(* IEC 61131-3 sources: Industry-PLC-LLM/data/PLCBEAD_repo/PLCBEAD_PLCEmbed-main/PLC-BEAD/Source/GEB/DWORD_OF_BYTE, 1 file *)

(* ---- DWORD_OF_BYTE.ST ---- *)
FUNCTION DWORD_OF_BYTE:DWORD
	VAR_INPUT
		B3 :	BYTE;
		B2 :	BYTE;
		B1 :	BYTE;
		B0 :	BYTE;
	END_VAR

	DWORD_OF_BYTE := SHL(SHL(SHL(BYTE_TO_DWORD(B3),8) OR BYTE_TO_DWORD(B2),8) OR BYTE_TO_DWORD(B1),8) OR BYTE_TO_DWORD(B0);

END_FUNCTION

PROGRAM program0
  VAR
    LocalVar0 : BYTE;
	LocalVaR1  : BYTE;
	LocalVaR2 : BYTE;
	LocalVar3 : BYTE;
	LocalOUT  : DWORD;
  END_VAR
  	LocalOUT := DWORD_OF_BYTE(LocalVar0, LocalVaR1 , LocalVaR2, LocalVar3);
END_PROGRAM
